TYPE ST_AxisStruct :
STRUCT
    stControl: ST_AxisControl;
    stStatus: ST_AxisStatus;
    stConfig: ST_AxisConfig;
    stError: ST_AxisError;
    stInputs: ST_AxisInputs;
    //The NC axis link to the hardware that is controlling
    Axis: AXIS_REF; (*~ (OPC: 0 : unavailable for OPC-clients) *)
END_STRUCT
END_TYPE

(* stored: Version 1.1.0.1, ProductVersion 3.1.4024.11
   DUT ST_AxisStruct: Id {9732127f-85ab-48d1-a591-d13402fe3665} *)
